FUNCTION_BLOCK FB_UnitTestTarget02 EXTENDS FB_Target
VAR_INPUT
END_VAR
VAR_OUTPUT
END_VAR
VAR
	fbTestsuite:			FB_Testsuite;				// Testsuite
	sValue:					STRING;
END_VAR

SUPER^();

fbTestsuite();


CASE fbTestsuite.P_Testcase OF
	E_Testcase.Init:
		sValue:= 'Test';

	E_Testcase.Start:
		// First test case
		fbTestsuite.P_Assert.M_Equals_STRING('Test', sValue, 'Check string value "Test"');
		fbTestsuite.M_Testcase('FB_Target', T#1S, '', '', 1);
		
	// secound test case
	1:
		fbTestsuite.P_Assert.M_IsTRUE('Test2' <> sValue, 'Check string value "Test2"');
		fbTestsuite.M_Testcase('FB_Target', T#1S, '', '', E_Testcase.Done);
		
	E_Testcase.Done:
		
END_CASE

METHOD FB_init : BOOL
VAR_INPUT
	bInitRetains : BOOL; // if TRUE, the retain variables are initialized (warm start / cold start)
	bInCopyCode : BOOL;  // if TRUE, the instance afterwards gets moved into the copy code (online change)
END_VAR
//// Add Testsuite to Testsuites
fbTestsuites.M_Add(fbTestsuite);
fbTestsuite.P_File:= 'FB_Target';
END_METHOD

END_FUNCTION_BLOCK

(* stored: Version 1.1.0.1
   POU FB_UnitTestTarget02: Id {8cae36d2-7866-0e80-1aad-bec70b8a78bb}, SpecialFunc None
   Method FB_init: Id {4878ff08-e607-0b76-3564-1b9a2e778b95} *)
